TYPE ST_ServiceCtrlBase :
STRUCT
	Start : BOOL;
	Reset : BOOL;
	Stop : BOOL;
	Abort : BOOL;
	Mode : T_PackMLMode;
END_STRUCT
END_TYPE

(* stored: Version 1.1.0.1, ProductVersion 3.1.4026.18
   DUT ST_ServiceCtrlBase: Id {205f631f-f425-47da-b81b-65944d80c767} *)
